(* PLC project Generated.project, CODESYS CODESYS V3.5 SP19 Patch 1 *)
(* stored: creationDateTime 2026-09-17T22:10:58.115402, modificationDateTime 2026-09-17T22:10:58.115402 *)

TYPE ST_Chain_Winch_Outputs : STRUCT
  Idx501_CmdRelayAscent_RQ : BOOL;  (* 1 = Relais Ascending ON | 0 = OFF *)
  Idx502_CmdRelayDescent_RQ : BOOL;  (* 1 = Relais Descending ON | 0 = OFF *)
  Idx503_CmdSpeedContactor1_DQ : BOOL;  (* 1 = Contacteur Vitesse 1 ON | 0 = OFF *)
  Idx504_CmdSpeedContactor4_DQ : BOOL;  (* 1 = Contacteur Vitesse 4 ON (Plein Gaz) | 0 = OFF *)
  Idx505_CmdBrakeRelease_RQ : BOOL;  (* 1 = Bobine Frein Alimentée (Ouvert) | 0 = Non Alimentée (Serré) *)
END_STRUCT;
END_TYPE
